Yaskawa INFORM job: YYYYYY.JBI

/JOB
//NAME YYYYYY
//POS
///NPOS 0,0,0,1,0,0
///TOOL 0
///POSTYPE BASE
///RECTAN
///RCONF 0,0,0,0,0,0,0,0,0,0,0,0,0,0,0,0,0,0,0,0,0,0,0,0
P00091=1.048,0.648,3.624,0.0000,0.0000,0.0000
//INST
///DATE 2024/11/05 16:32
///ATTR SC,RW,RJ
////FRAME ROBOT
///GROUP1 RB1,BS1
///GROUP2 ST1
NOP
SFTON P091
END
